// TIA Portal project "Server_Client_Test" (V15.1)

(* hardware
DEVICE "S71500/ET200MP-Station_1"  S7-1500 station
   slot 0: "Profilschiene_0"  Rack  6ES7 590-1***0-0AA0
   slot 1: "PLC_1"  CPU 1518-4 PN/DP MFP  6ES7 518-4AX00-1AB0  V2.6
      slot 3: "CPU-Display_1"  6ES7591-1BA00-0AA0
*)

// ===== PLC "PLC_1"  CPU 1518-4 PN/DP MFP =====

DATA_BLOCK "Send"   // DB1
{ S7_Optimized_Access := 'FALSE' }
VERSION : 0.1
   VAR
      Send_Data : Byte;
   END_VAR
BEGIN
END_DATA_BLOCK

DATA_BLOCK "RCV"   // DB2
{ S7_Optimized_Access := 'FALSE' }
VERSION : 0.1
   VAR
      RCV_Data : Byte;
   END_VAR
BEGIN
END_DATA_BLOCK

// folder: System blocks/Program resources

DATA_BLOCK "PLC_1_Send_DB"   // DB5
{ S7_Optimized_Access := 'TRUE' }
AUTHOR : SIMATIC
FAMILY : MC7Plus
NAME : TC_IP_v4
VERSION : 1.0
// stored: InstanceOfName TCON_IP_v4
"TCON_IP_v4"
BEGIN
   ID := 1;
   InterfaceId := 64;
   RemotePort := 2710;
   ActiveEstablished := true;
   RemoteAddress.ADDR[1] := 192;
   RemoteAddress.ADDR[2] := 168;
   RemoteAddress.ADDR[4] := 169;
END_DATA_BLOCK

DATA_BLOCK "PLC_1_Receive_DB_1"   // DB7
{ S7_Optimized_Access := 'TRUE' }
AUTHOR : SIMATIC
FAMILY : MC7Plus
NAME : TC_IP_v4
VERSION : 1.0
// stored: InstanceOfName TCON_IP_v4
"TCON_IP_v4"
BEGIN
   ID := 3;
   InterfaceId := 64;
   LocalPort := 2700;
END_DATA_BLOCK

// folder: (top level)

ORGANIZATION_BLOCK "Main"   // OB1, FBD, ProgramCycle
TITLE = "Main Program Sweep (Cycle)"
{ S7_Optimized_Access := 'TRUE' }
VERSION : 0.1
   VAR_INPUT
      Initial_Call : Bool;   // Initial call of this OB
      Remanence : Bool;   // =True, if remanent data are available
   END_VAR
BEGIN

REGION Network 1
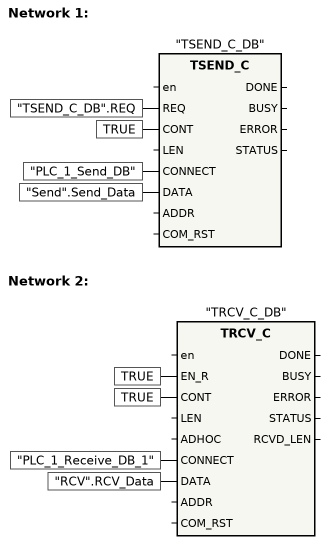
   "TSEND_C_DB"(REQ := "TSEND_C_DB".REQ, CONT := TRUE, CONNECT := "PLC_1_Send_DB", DATA := "Send".Send_Data);   // TSEND_C
END_REGION

REGION Network 2
   "TRCV_C_DB"(EN_R := TRUE, CONT := TRUE, CONNECT := "PLC_1_Receive_DB_1", DATA := "RCV".RCV_Data);   // TRCV_C
END_REGION
END_ORGANIZATION_BLOCK